Xinje XCPPro project, PLC1: XC3-24 (software 3.3L)

PROGRAM Ladder

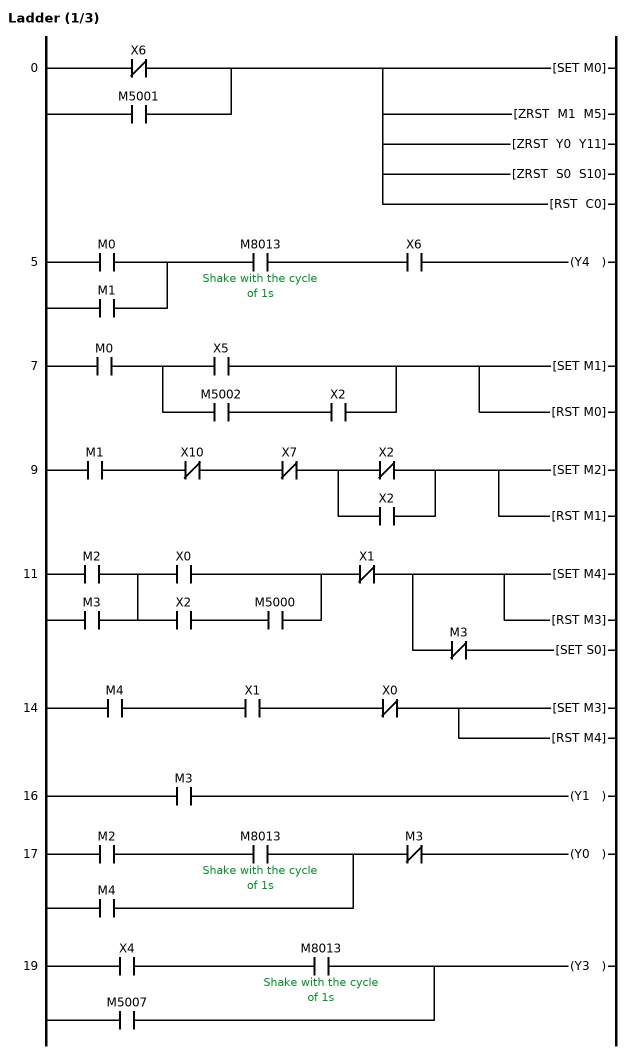
LDI    X6
OR     M5001
SET    M0
ZRST   M1 M5
ZRST   Y0 Y11
ZRST   S0 S10
RST    C0
LD     M0
OR     M1
AND    M8013	; Shake with the cycle of 1s
AND    X6
OUT    Y4
LD     M0
LD     X5
LD     M5002
AND    X2
ORB
ANB
SET    M1
RST    M0
LD     M1
ANI    X10
ANI    X7
LDI    X2
OR     X2
ANB
SET    M2
RST    M1
LD     M2
OR     M3
LD     X0
LD     X2
AND    M5000
ORB
ANB
ANI    X1
SET    M4
RST    M3
ANI    M3
SET    S0
LD     M4
AND    X1
ANI    X0
SET    M3
RST    M4
LD     M3
OUT    Y1
LD     M2
AND    M8013	; Shake with the cycle of 1s
OR     M4
ANI    M3
OUT    Y0
LD     X4
AND    M8013	; Shake with the cycle of 1s
OR     M5007
OUT    Y3

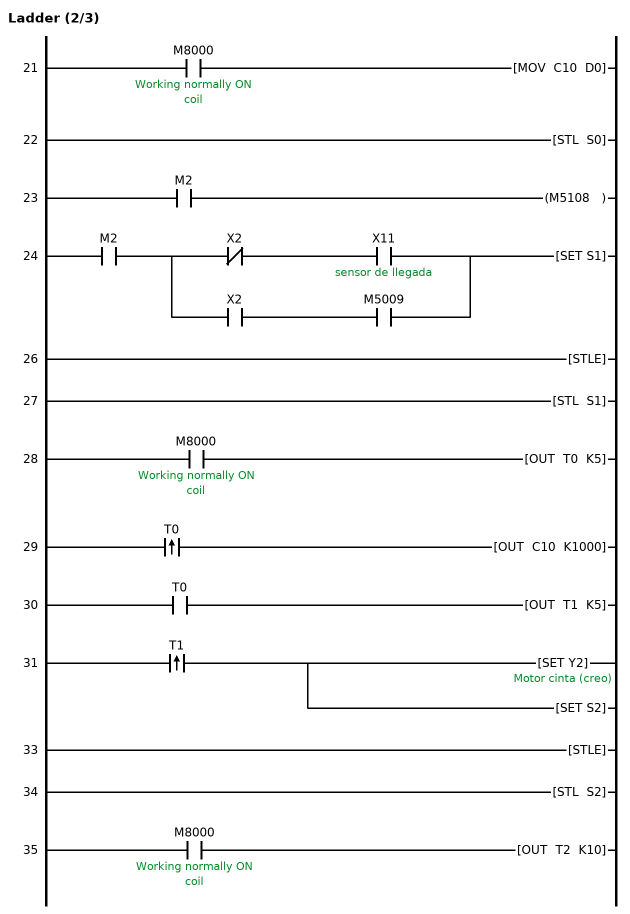
LD     M8000	; Working normally ON coil
MOV    C10 D0
STL    S0
LD     M2
OUT    M5108
LD     M2
LDI    X2
AND    X11	; sensor de llegada
LD     X2
AND    M5009
ORB
ANB
SET    S1
STLE
STL    S1
LD     M8000	; Working normally ON coil
OUT    T0 K5
LDP    T0
OUT    C10 K1000
LD     T0
OUT    T1 K5
LDP    T1
SET    Y2	; Motor cinta (creo)
SET    S2
STLE
STL    S2
LD     M8000	; Working normally ON coil
OUT    T2 K10

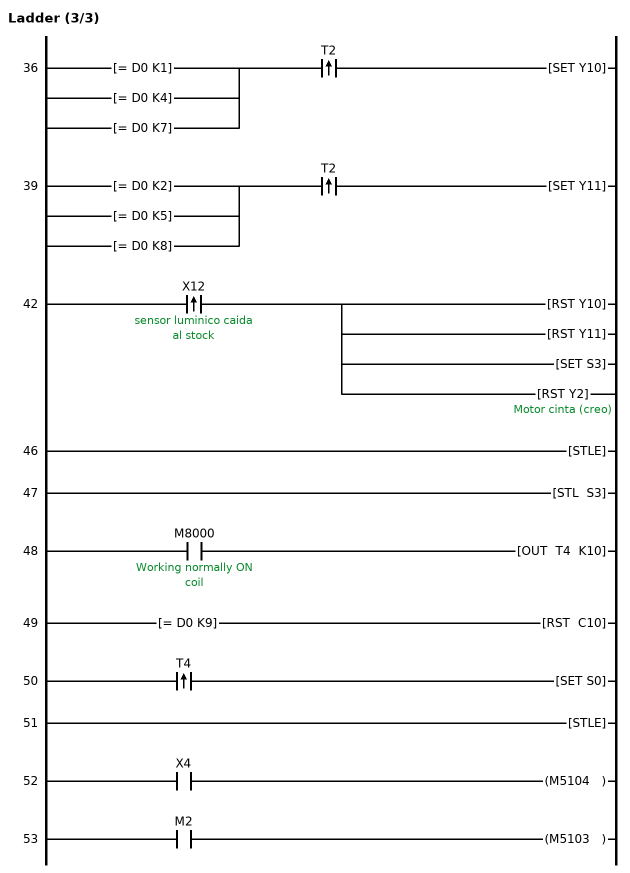
LD=    D0 K1
OR=    D0 K4
OR=    D0 K7
ANDP   T2
SET    Y10
LD=    D0 K2
OR=    D0 K5
OR=    D0 K8
ANDP   T2
SET    Y11
LDP    X12	; sensor luminico caida al stock
RST    Y10
RST    Y11
SET    S3
RST    Y2	; Motor cinta (creo)
STLE
STL    S3
LD     M8000	; Working normally ON coil
OUT    T4 K10
LD=    D0 K9
RST    C10
LDP    T4
SET    S0
STLE
LD     X4
OUT    M5104
LD     M2
OUT    M5103